// function block for reed switch with the option of debouncing + rising and falling edge detection.
FUNCTION_BLOCK FB_Component_ReedSwitch IMPLEMENTS I_Component
VAR_INPUT
	bRawSignal		: BOOL;				// Raw input sensor
	tDebounce		: TIME := T#0MS;	// Debounce time
	tTimeout		: TIME := T#0MS;
	
	sName			: STRING[20];
	bEnable     	: BOOL;
END_VAR

VAR_OUTPUT
	bSensorActive	: BOOL;
	bTimeout		: BOOL;
	eState			: E_ComponentState;
	sStatusText 	: STRING[100];
END_VAR

VAR
	tDebounceTimer	: TON;
	tTimeoutTimer	: TON;
	
	bLastStableSignal: BOOL;
	bPendingSignal: BOOL;
END_VAR

tDebounceTimer.PT 	:= tDebounce;
tTimeoutTimer.PT	:= tTimeout;

IF bEnable THEN
	CASE eState OF
		E_ComponentState.READY: 	IF bRawSignal <> bLastStableSignal THEN
										bPendingSignal := bRawSignal;
										eState := E_ComponentState.BUSY;
									ELSE
										tTimeoutTimer(IN := FALSE);
										tDebounceTimer(IN := FALSE);
									END_IF
									sStatusText := 'sensor active';
		
		E_ComponentState.BUSY:		tDebounceTimer(IN := TRUE);
									IF bRawSignal <> bPendingSignal THEN			// if signal bounces go back to ready state	
										eState := E_ComponentState.DONE;
									END_IF
			
									IF tDebounceTimer.Q THEN						// if signal stays stable for debounce duration -> trigger timeout
										eState := E_ComponentState.TIMEOUT;
									END_IF
									sStatusText := 'Debouncing sensor';
									
		E_ComponentState.TIMEOUT:	tTimeoutTimer(IN := TRUE);
									bLastStableSignal := bPendingSignal;			// output stable signal
									bSensorActive := bLastStableSignal;
									IF tTimeoutTimer.Q THEN
										eState := E_ComponentState.DONE;
									END_IF
									sStatusText := 'sensor timeout';
			
		E_ComponentState.DONE:		tTimeoutTimer(IN := FALSE);
									tDebounceTimer(IN := FALSE);
	END_CASE
END_IF

METHOD M_Halt : BOOL
VAR_INPUT
END_VAR
tDebounceTimer(IN := FALSE);
eState := E_ComponentState.HALTED;
END_METHOD

METHOD M_Start : BOOL
VAR_INPUT
END_VAR
IF eState <> E_ComponentState.BUSY AND eState <> E_ComponentState.TIMEOUT THEN
	eState := E_ComponentState.READY;
END_IF;
END_METHOD

METHOD M_Stop : BOOL
VAR_INPUT
END_VAR
IF eState <> E_ComponentState.BUSY AND eState <> E_ComponentState.TIMEOUT  THEN
	eState := E_ComponentState.DONE;
END_IF
END_METHOD

END_FUNCTION_BLOCK

(* stored: Version 1.1.0.1, ProductVersion 3.1.4024.15
   POU FB_Component_ReedSwitch: Id {f639b4a8-9d3e-46fd-a4ee-568d4dd5739a}, SpecialFunc None
   Method M_Halt: Id {c94396e9-4b2a-428e-b504-c709afbc748b}
   Method M_Start: Id {3ee6110b-c203-4bb9-9caa-b0b18392f854}
   Method M_Stop: Id {60cdd494-a322-4122-a75f-cf6898b5dc26} *)
